(* IEC 61131-3 sources: cc_kush_rewrite/Library, 11 files *)

(* ---- FB_AnalogInput.st ---- *)
FUNCTION_BLOCK FB_AnalogInput
VAR_INPUT
    // Основные входы
    xSimulation     : BOOL;             // Флаг симуляции
    iADC_Code       : INT;              // Код АЦП от модуля аналогового входа
    refEngValue     : REFERENCE TO REAL; // Ссылка на переменную в инженерных единицах
    refSimValue     : REFERENCE TO REAL; // Ссылка на переменную для ручного задания в симуляции

    // Параметры уставок по току (4-20 мА)
    rAlarm_LL       : REAL := 1.1852;      // Аварийно низкий уровень тока (мА)
    rAlarm_L        : REAL := 3.9995;      // Низкий уровень тока (мА)
    rAlarm_H        : REAL := 20.0005;     // Высокий уровень тока (мА)
    rAlarm_HH       : REAL := 22.81;       // Аварийно высокий уровень тока (мА)

    // Параметры АЦП
    iADC_Max        : INT := 32767;     // Максимальный код АЦП
    iADC_Min        : INT := 0;         // Минимальный код АЦП

    // Параметры масштабирования
    rEngValue_Max   : REAL := 100.0;    // Максимальное значение в ед. измерения
    rEngValue_Min   : REAL := 0.0;      // Минимальное значение в ед. измерения

    // Параметры тока
    rCurrent_Max    : REAL := 20.0;     // Максимальный ток (мА)
    rCurrent_Min    : REAL := 4.0;      // Минимальный ток (мА)
END_VAR

VAR_OUTPUT
    // Выходы
    rCurrent_mA     : REAL;             // Ток 4-20 мА

    // Тревоги по току
    xAlarm_LL       : BOOL;             // Аварийно низкий уровень
    xAlarm_L        : BOOL;             // Низкий уровень
    xAlarm_H        : BOOL;             // Высокий уровень
    xAlarm_HH       : BOOL;             // Аварийно высокий уровень
	eAlarmStatus : E_AlarmSetpoints;
END_VAR

VAR
    rScaledValue    : REAL;             // Внутреннее масштабированное значение
    rADC_Range      : REAL;             // Диапазон АЦП
    rEng_Range      : REAL;             // Диапазон инженерных единиц
    rCurrent_Range  : REAL;             // Диапазон тока
    _xSimulation_Prev : BOOL;           // Предыдущее состояние симуляции (для детектирования фронта)
END_VAR

// Расчёт диапазонов
rADC_Range := INT_TO_REAL(iADC_Max - iADC_Min);
rEng_Range := rEngValue_Max - rEngValue_Min;
rCurrent_Range := rCurrent_Max - rCurrent_Min;

// Защита от деления на ноль
IF rADC_Range = 0.0 THEN
    rADC_Range := 1.0;
END_IF

// Масштабирование кода АЦП в ток 4-20 мА
rCurrent_mA := rCurrent_Min +
               (INT_TO_REAL(iADC_Code - iADC_Min) / rADC_Range) * rCurrent_Range;

// Логика симуляции и масштабирования
IF xSimulation THEN
    // Режим симуляции активен

    // При переходе в режим симуляции (rising edge) - инициализировать симуляцию
    IF NOT _xSimulation_Prev AND __ISVALIDREF(refEngValue) AND __ISVALIDREF(refSimValue) THEN
        // Однократно передать текущее значение в переменную симуляции
        refSimValue := refEngValue;
    END_IF

    // В режиме симуляции - использовать значение из переменной симуляции
    IF __ISVALIDREF(refEngValue) AND __ISVALIDREF(refSimValue) THEN
        refEngValue := refSimValue;
    END_IF

ELSE
    // Режим симуляции выключен - работает обычное масштабирование
    IF __ISVALIDREF(refEngValue) THEN
        rScaledValue := rEngValue_Min +
                        ((rCurrent_mA - rCurrent_Min) / rCurrent_Range) * rEng_Range;
        refEngValue := rScaledValue;
    END_IF
END_IF

// Сохранить текущее состояние симуляции для следующего цикла
_xSimulation_Prev := xSimulation;

// Обработка тревог по току
// Аварийно низкий уровень (обрыв линии)
xAlarm_LL := rCurrent_mA < rAlarm_LL;

// Низкий уровень
xAlarm_L := (rCurrent_mA >= rAlarm_LL) AND (rCurrent_mA < rAlarm_L);

// Высокий уровень
xAlarm_H := (rCurrent_mA > rAlarm_H) AND (rCurrent_mA <= rAlarm_HH);

// Аварийно высокий уровень (перегрузка)
xAlarm_HH := rCurrent_mA > rAlarm_HH;

// Обновление общего статуса тревоги (по приоритету)
IF xAlarm_LL THEN
    eAlarmStatus := E_AlarmSetpoints.LL;
ELSIF xAlarm_HH THEN
    eAlarmStatus := E_AlarmSetpoints.HH;
ELSIF xAlarm_L THEN
    eAlarmStatus := E_AlarmSetpoints.L;
ELSIF xAlarm_H THEN
    eAlarmStatus := E_AlarmSetpoints.H;
ELSE
    eAlarmStatus := E_AlarmSetpoints.Normal;
END_IF

END_FUNCTION_BLOCK

(* ---- FB_AnalogOutput.st ---- *)
FUNCTION_BLOCK FB_AnalogOutput
VAR_INPUT
    // Основные входы
    xEnable         : BOOL := TRUE;     // Разрешение работы выхода
    rEngValue       : REAL;             // Значение в инженерных единицах для вывода

    // Параметры масштабирования
    rEngValue_Max   : REAL := 100.0;    // Максимальное значение в ед. измерения
    rEngValue_Min   : REAL := 0.0;      // Минимальное значение в ед. измерения

    // Параметры тока
    rCurrent_Max    : REAL := 20.0;     // Максимальный ток (мА)
    rCurrent_Min    : REAL := 4.0;      // Минимальный ток (мА)

    // Параметры АЦП (DAC)
    iDAC_Max        : INT := 32767;     // Максимальный код АЦП
    iDAC_Min        : INT := 0;         // Минимальный код АЦП

    // Параметры уставок по току (4-20 мА)
    rAlarm_LL       : REAL := 1.1852;      // Аварийно низкий уровень тока (мА)
    rAlarm_L        : REAL := 3.9995;      // Низкий уровень тока (мА)
    rAlarm_H        : REAL := 20.0005;     // Высокий уровень тока (мА)
    rAlarm_HH       : REAL := 22.81;       // Аварийно высокий уровень тока (мА)

    // Опции
    xEnableClamp    : BOOL := TRUE;     // Включить ограничение выхода за пределы диапазона
END_VAR

VAR_OUTPUT
    // Выходы
    rCurrent_mA     : REAL;             // Выходной ток 4-20 мА
    iDAC_Code       : INT;              // Код АЦП для модуля аналогового выхода

    // Тревоги по току
    xAlarm_LL       : BOOL;             // Аварийно низкий уровень
    xAlarm_L        : BOOL;             // Низкий уровень
    xAlarm_H        : BOOL;             // Высокий уровень
    xAlarm_HH       : BOOL;             // Аварийно высокий уровень
    eAlarmStatus    : E_AlarmSetpoints; // Общий статус тревоги

    // Диагностика диапазона
    xOverRange      : BOOL;             // Превышение верхнего предела
    xUnderRange     : BOOL;             // Выход за нижний предел
    xOutOfRange     : BOOL;             // Общий флаг выхода за пределы
END_VAR

VAR
    rEng_Range      : REAL;             // Диапазон инженерных единиц
    rCurrent_Range  : REAL;             // Диапазон тока
    rDAC_Range      : REAL;             // Диапазон АЦП
    rNormalizedValue : REAL;            // Нормализованное значение (0.0 - 1.0)
    rEngValue_Clamped : REAL;           // Ограниченное значение в инженерных единицах
END_VAR

// Расчёт диапазонов
rEng_Range := rEngValue_Max - rEngValue_Min;
rCurrent_Range := rCurrent_Max - rCurrent_Min;
rDAC_Range := INT_TO_REAL(iDAC_Max - iDAC_Min);

// Защита от деления на ноль
IF rEng_Range = 0.0 THEN
    rEng_Range := 1.0;
END_IF

// Проверка выхода за пределы
xUnderRange := rEngValue < rEngValue_Min;
xOverRange := rEngValue > rEngValue_Max;
xOutOfRange := xUnderRange OR xOverRange;

// Ограничение значения (если включено)
IF xEnableClamp THEN
    IF rEngValue < rEngValue_Min THEN
        rEngValue_Clamped := rEngValue_Min;
    ELSIF rEngValue > rEngValue_Max THEN
        rEngValue_Clamped := rEngValue_Max;
    ELSE
        rEngValue_Clamped := rEngValue;
    END_IF
ELSE
    rEngValue_Clamped := rEngValue;
END_IF

// Нормализация значения (0.0 - 1.0)
rNormalizedValue := (rEngValue_Clamped - rEngValue_Min) / rEng_Range;

// Преобразование в ток 4-20 мА
rCurrent_mA := rCurrent_Min + rNormalizedValue * rCurrent_Range;

// Преобразование в код АЦП
IF xEnable THEN
    iDAC_Code := iDAC_Min + REAL_TO_INT(rNormalizedValue * rDAC_Range);
ELSE
    // Если выход отключен - безопасное значение (минимальный ток)
    iDAC_Code := iDAC_Min;
    rCurrent_mA := rCurrent_Min;
END_IF

// Обработка тревог по току
// Аварийно низкий уровень
xAlarm_LL := rCurrent_mA < rAlarm_LL;

// Низкий уровень
xAlarm_L := (rCurrent_mA >= rAlarm_LL) AND (rCurrent_mA < rAlarm_L);

// Высокий уровень
xAlarm_H := (rCurrent_mA > rAlarm_H) AND (rCurrent_mA <= rAlarm_HH);

// Аварийно высокий уровень
xAlarm_HH := rCurrent_mA > rAlarm_HH;

// Обновление общего статуса тревоги (по приоритету)
IF xAlarm_LL THEN
    eAlarmStatus := E_AlarmSetpoints.LL;
ELSIF xAlarm_HH THEN
    eAlarmStatus := E_AlarmSetpoints.HH;
ELSIF xAlarm_L THEN
    eAlarmStatus := E_AlarmSetpoints.L;
ELSIF xAlarm_H THEN
    eAlarmStatus := E_AlarmSetpoints.H;
ELSE
    eAlarmStatus := E_AlarmSetpoints.Normal;
END_IF

END_FUNCTION_BLOCK

(* ---- FB_FrequencyControl.st ---- *)
FUNCTION_BLOCK FB_FrequencyControl
VAR_INPUT
    irMaxFrequency : REAL := 100.0;             // Максимальная частота
    irStep : REAL := 1.0;                       // Шаг изменения частоты по умолчанию
    rTargetFrequency : REAL := 0.0;             // Целевая частота (уставка)
    xPulse : BOOL;                              // Импульсный сигнал для вычисления
    xConditionToProceed : BOOL := TRUE;         // Условия для продолжения вычисления
    xReset : BOOL;                              // Сброс частоты в ноль
    xHold : BOOL;                               // Удержание текущей частоты
END_VAR
VAR_OUTPUT
    qrCurrentFrequency : REAL;                  // Текущая выходная частота
    qrTargetFrequency : REAL;                   // Целевая частота
    qxTargetReached : BOOL;                     // Флаг достижения целевой частоты
END_VAR
VAR
    _rSetFrequency : REAL;                      // Целевая частота (уставка) внутренняя
    _rCurrentFrequency : REAL;                  // Текущая частота (внутренняя)
    _xInitialized : BOOL := FALSE;              // Флаг инициализации
END_VAR

// Инициализация при первом вызове
IF NOT _xInitialized THEN
    _rCurrentFrequency := 0.0;
    _rSetFrequency := 0.0;
    _xInitialized := TRUE;
END_IF

// Сброс частоты
IF xReset THEN
    _rCurrentFrequency := 0.0;
    _rSetFrequency := 0.0;
    qrCurrentFrequency := 0.0;
    qrTargetFrequency := 0.0;
    qxTargetReached := TRUE;
    RETURN;
END_IF

// Удержание текущей частоты
IF xHold THEN
    _rSetFrequency := _rCurrentFrequency;
    qxTargetReached := TRUE;
END_IF

// Обновление целевой частоты
_rSetFrequency := rTargetFrequency;

// Ограничение целевой частоты
IF _rSetFrequency > irMaxFrequency THEN
    _rSetFrequency := irMaxFrequency;
ELSIF _rSetFrequency < 0.0 THEN
    _rSetFrequency := 0.0;
END_IF

// Обработка изменения частоты
IF xPulse AND xConditionToProceed THEN
    // Плавное изменение частоты к уставке
    IF _rCurrentFrequency < _rSetFrequency - irStep THEN
        // Увеличиваем частоту
        _rCurrentFrequency := _rCurrentFrequency + irStep;
        qxTargetReached := FALSE;
    ELSIF _rCurrentFrequency > _rSetFrequency + irStep THEN
        // Уменьшаем частоту
        _rCurrentFrequency := _rCurrentFrequency - irStep;
        qxTargetReached := FALSE;
    ELSE
        // Достигли целевой частоты
        _rCurrentFrequency := _rSetFrequency;
        qxTargetReached := TRUE;
    END_IF
ELSE
    // Проверяем, достигнута ли целевая частота
    IF ABS(_rCurrentFrequency - _rSetFrequency) < 0.01 THEN
        qxTargetReached := TRUE;
    ELSE
        qxTargetReached := FALSE;
    END_IF
END_IF

// Обновляем выходные значения
qrCurrentFrequency := _rCurrentFrequency;
qrTargetFrequency := _rSetFrequency;

END_FUNCTION_BLOCK

(* ---- FB_NumericChangeDetector.st ---- *)
FUNCTION_BLOCK FB_NumericChangeDetector
VAR_INPUT
    irValue : REAL;                             // Входное числовое значение для мониторинга
    xReset : BOOL;                              // Сброс детектора изменений
END_VAR
VAR_OUTPUT
    qxChangeDetected : BOOL;                    // Импульс при обнаружении изменения значения
    qrCurrentValue : REAL;                      // Текущее отслеживаемое значение
    qrPreviousValue : REAL;                     // Предыдущее значение
    qrValueDifference : REAL;                   // Разность между текущим и предыдущим значением
    qxValueIncreased : BOOL;                    // Флаг увеличения значения
    qxValueDecreased : BOOL;                    // Флаг уменьшения значения
END_VAR
VAR
    _rPreviousValue : REAL := 0.0;              // Предыдущее значение для сравнения
    _xFirstCycle : BOOL := TRUE;                // Флаг первого цикла выполнения
    _rt_Change : R_TRIG;                        // Триггер для генерации импульса
    _xValueChanged : BOOL := FALSE;             // Внутренний флаг изменения
END_VAR

// Сброс детектора
IF xReset THEN
    _rPreviousValue := irValue;
    _xFirstCycle := TRUE;
    _xValueChanged := FALSE;
    _rt_Change(CLK := FALSE);
    qxChangeDetected := FALSE;
    qrValueDifference := 0.0;
    qxValueIncreased := FALSE;
    qxValueDecreased := FALSE;
    RETURN;
END_IF

// Пропускаем первый цикл для корректной инициализации
IF _xFirstCycle THEN
    _rPreviousValue := irValue;
    _xFirstCycle := FALSE;
    _xValueChanged := FALSE;
ELSE
    // Проверяем изменение значения
    IF _rPreviousValue <> irValue THEN
        _xValueChanged := TRUE;
    ELSE
        _xValueChanged := FALSE;
    END_IF
END_IF

// Генерируем импульс при изменении через R_TRIG
_rt_Change(CLK := _xValueChanged);
qxChangeDetected := _rt_Change.Q;

// Вычисляем разность
qrValueDifference := irValue - _rPreviousValue;

// Определяем направление изменения
qxValueIncreased := _xValueChanged AND (irValue > _rPreviousValue);
qxValueDecreased := _xValueChanged AND (irValue < _rPreviousValue);

// Обновляем предыдущее значение после всех вычислений
IF _xValueChanged THEN
    _rPreviousValue := irValue;
END_IF

// Обновляем выходы
qrCurrentValue := irValue;
qrPreviousValue := _rPreviousValue;

END_FUNCTION_BLOCK

(* ---- FB_PreStartAlarm.st ---- *)
FUNCTION_BLOCK FB_PreStartAlarm
VAR_INPUT
    ixStart : BOOL;                    // Сигнал на запуск
    ixStop : BOOL;                     // Сигнал на стоп (Reset)
    itFirstSignal : TIME;              // Уставка первого сигнала
    itPauseAfterFirst : TIME;          // Уставка паузы после первого сигнала
    itSecondSignal : TIME;             // Уставка второго сигнала
    itPauseAfterSecond : TIME;         // Уставка паузы после второго сигнала
END_VAR

VAR_OUTPUT
    qxAlarmPower : BOOL;               // Питание звуковой сигнализации
    qxActive : BOOL;                   // Активная работа ФБ
    qxComplete : BOOL;                 // Импульс о завершении работы
    qnSecondsRemaining : INT;          // Количество секунд до завершения
    qwSecondsRemaining : WORD;		    // Количество секунд до завершения (тип WORD)
END_VAR

VAR
    _eState : (
        IDLE := 0,              // Ожидание запуска
        FIRST_SIGNAL := 1,      // Первый звуковой сигнал
        PAUSE_AFTER_FIRST := 2, // Пауза после первого сигнала
        SECOND_SIGNAL := 3,     // Второй звуковой сигнал
        PAUSE_AFTER_SECOND := 4,// Пауза после второго сигнала
        COMPLETE := 5           // Завершение
    ) := IDLE;                         // Состояние автомата
    _tonTimer : TON;                   // Универсальный таймер для всех этапов
    _xCompleteInternal : BOOL;         // Внутренний сигнал завершения
    _rtrigComplete : R_TRIG;           // Детектор переднего фронта для импульса завершения
END_VAR

qwSecondsRemaining := TO_WORD(qnSecondsRemaining);

// Обработка сигнала СТОП (сброс)
IF ixStop THEN
    _eState := IDLE;
    qxActive := FALSE;
    qxAlarmPower := FALSE;
    _tonTimer(IN := FALSE);
    _xCompleteInternal := FALSE;
    qxComplete := FALSE;
    qnSecondsRemaining := 0;
    RETURN;
END_IF

// Автомат состояний
CASE _eState OF

    IDLE: // Ожидание запуска
        qxActive := FALSE;
        qxAlarmPower := FALSE;
        _xCompleteInternal := FALSE;
        _tonTimer(IN := FALSE);
        qnSecondsRemaining := 0;

        IF ixStart THEN
			qxActive := TRUE;
            _eState := FIRST_SIGNAL;
        END_IF

    FIRST_SIGNAL: // Первый сигнал
        qxAlarmPower := TRUE;
        _tonTimer(IN := TRUE, PT := itFirstSignal);

        // Расчет оставшегося времени в секундах
        qnSecondsRemaining := DINT_TO_INT(
            (TIME_TO_DINT(itFirstSignal - _tonTimer.ET) +
             TIME_TO_DINT(itPauseAfterFirst) +
             TIME_TO_DINT(itSecondSignal) +
             TIME_TO_DINT(itPauseAfterSecond)) / 1000
        );

        IF _tonTimer.Q THEN
            _tonTimer(IN := FALSE);
            _eState := PAUSE_AFTER_FIRST;
        END_IF

    PAUSE_AFTER_FIRST: // Пауза после первого сигнала
        qxAlarmPower := FALSE;
        _tonTimer(IN := TRUE, PT := itPauseAfterFirst);

        // Расчет оставшегося времени в секундах
        qnSecondsRemaining := DINT_TO_INT(
            (TIME_TO_DINT(itPauseAfterFirst - _tonTimer.ET) +
             TIME_TO_DINT(itSecondSignal) +
             TIME_TO_DINT(itPauseAfterSecond)) / 1000
        );

        IF _tonTimer.Q THEN
            _tonTimer(IN := FALSE);
            _eState := SECOND_SIGNAL;
        END_IF

    SECOND_SIGNAL: // Второй сигнал
        qxAlarmPower := TRUE;
        _tonTimer(IN := TRUE, PT := itSecondSignal);

        // Расчет оставшегося времени в секундах
        qnSecondsRemaining := DINT_TO_INT(
            (TIME_TO_DINT(itSecondSignal - _tonTimer.ET) +
             TIME_TO_DINT(itPauseAfterSecond)) / 1000
        );

        IF _tonTimer.Q THEN
            _tonTimer(IN := FALSE);
            _eState := PAUSE_AFTER_SECOND;
        END_IF

    PAUSE_AFTER_SECOND: // Пауза после второго сигнала
        qxAlarmPower := FALSE;
        _tonTimer(IN := TRUE, PT := itPauseAfterSecond);

        // Расчет оставшегося времени в секундах
        qnSecondsRemaining := DINT_TO_INT(
            TIME_TO_DINT(itPauseAfterSecond - _tonTimer.ET) / 1000
        );

        IF _tonTimer.Q THEN
            _tonTimer(IN := FALSE);
            _eState := COMPLETE;
        END_IF

    COMPLETE: // Завершение
        qxAlarmPower := FALSE;
        qxActive := FALSE;
        _xCompleteInternal := TRUE;
        qnSecondsRemaining := 0;
        _eState := IDLE;  // Вернуться в начальное состояние
END_CASE

// Генерация импульса завершения через R_TRIG
_rtrigComplete(CLK := _xCompleteInternal);
qxComplete := _rtrigComplete.Q;

END_FUNCTION_BLOCK

(* ---- FB_ProportionPID.st ---- *)
FUNCTION_BLOCK FB_ProportionPID

// ============================================================================
// ВХОДНЫЕ ПЕРЕМЕННЫЕ
// ============================================================================
VAR_INPUT
    // ------------------------------------------------------------------------
    // Команды управления
    // ------------------------------------------------------------------------
    xEnable                 : BOOL;         // Разрешение работы блока
    xReset                  : BOOL;         // Сброс интегральной составляющей ПИД

    // ------------------------------------------------------------------------
    // Целевые пропорции (уставки оператора)
    // ------------------------------------------------------------------------
    rProportionTarget_1     : REAL;         // Целевая пропорция бункера 1 [0..1]
    rProportionTarget_2     : REAL;         // Целевая пропорция бункера 2 [0..1]
    rProportionTarget_3     : REAL;         // Целевая пропорция бункера 3 [0..1]
                                            // Сумма должна = 1.0 (100%)
                                            // Значение 0.0 = бункер неактивен

    // ------------------------------------------------------------------------
    // Фактические пропорции (с конвейерных весов)
    // ------------------------------------------------------------------------
    rProportionActual_1     : REAL;         // Фактическая пропорция бункера 1 [0..1]
    rProportionActual_2     : REAL;         // Фактическая пропорция бункера 2 [0..1]
    rProportionActual_3     : REAL;         // Фактическая пропорция бункера 3 [0..1]

    // ------------------------------------------------------------------------
    // Параметры ПИД-регулятора
    // ------------------------------------------------------------------------
    rPID_Kp                 : REAL := 1.0;  // Пропорциональный коэффициент
    rPID_Ki                 : REAL := 0.2;  // Интегральный коэффициент
    rPID_Kd                 : REAL := 0.05; // Дифференциальный коэффициент
    rPID_IntegralLimit      : REAL := 10.0; // Ограничение интеграла (anti-windup)
    rPID_DerivativeFilter   : REAL := 0.1;  // Коэффициент фильтрации D-составляющей [0..1]
                                            // 0 = нет фильтрации, 1 = максимум фильтра

    // ------------------------------------------------------------------------
    // Базовые частоты (рассчитываются заранее в INIT)
    // ------------------------------------------------------------------------
    rFrequencyBase_1        : REAL;         // Базовая частота бункера 1, Гц
    rFrequencyBase_2        : REAL;         // Базовая частота бункера 2, Гц
    rFrequencyBase_3        : REAL;         // Базовая частота бункера 3, Гц

    // ------------------------------------------------------------------------
    // Параметры оборудования
    // ------------------------------------------------------------------------
    rFrequency_Min          : REAL := 1.0;  // Минимальная частота ЧРП, Гц
    rFrequency_Max          : REAL := 35.0; // Максимальная частота ЧРП, Гц
    rFrequency_TargetSum    : REAL := 90.0; // Целевая суммарная частота для нормализации, Гц

    // ------------------------------------------------------------------------
    // Параметры расчета
    // ------------------------------------------------------------------------
    rDeltaTime              : REAL := 2;  // Период вызова блока, сек

    // ------------------------------------------------------------------------
    // Параметры алгоритма
    // ------------------------------------------------------------------------
    rScaleLimit_Min         : REAL := 0.1;  // Минимальный коэффициент масштабирования
    rScaleLimit_Max         : REAL := 3.0;  // Максимальный коэффициент масштабирования
    rProportionThreshold    : REAL := 0.001; // Порог для определения неактивного бункера
END_VAR

// ============================================================================
// ВЫХОДНЫЕ ПЕРЕМЕННЫЕ
// ============================================================================
VAR_OUTPUT
    // ------------------------------------------------------------------------
    // Управляющие воздействия (частоты ЧРП)
    // ------------------------------------------------------------------------
    qrFrequency_1           : REAL;         // Уставка частоты ЧРП бункера 1, Гц
    qrFrequency_2           : REAL;         // Уставка частоты ЧРП бункера 2, Гц
    qrFrequency_3           : REAL;         // Уставка частоты ЧРП бункера 3, Гц

    // ------------------------------------------------------------------------
    // Состояние работы
    // ------------------------------------------------------------------------
    qxActive                : BOOL;         // Блок активен и регулирует частоты
    qxError                 : BOOL;         // Ошибка работы блока
    quErrorCode             : UINT;         // Код ошибки:
                                            // 0 = нет ошибок
                                            // 1 = сумма пропорций = 0
                                            // 2 = неверный DeltaTime
                                            // 3 = неверные пределы частот
                                            // 4 = неверная целевая сумма частот

    // ------------------------------------------------------------------------
    // Диагностическая информация
    // ------------------------------------------------------------------------
    qrFrequency_Sum         : REAL;         // Фактическая суммарная частота, Гц
    qrProportionSum         : REAL;         // Сумма целевых пропорций
    qxProportionNormalized  : BOOL;         // TRUE = пропорции автоматически нормализованы

    // ------------------------------------------------------------------------
    // Выходы ПИД-регуляторов (для диагностики)
    // ------------------------------------------------------------------------
    qrPID_Output_1          : REAL;         // Выход ПИД регулятора 1 [0..1]
    qrPID_Output_2          : REAL;         // Выход ПИД регулятора 2 [0..1]
    qrPID_Output_3          : REAL;         // Выход ПИД регулятора 3 [0..1]

    qrPID_Error_1           : REAL;         // Текущая ошибка ПИД 1
    qrPID_Error_2           : REAL;         // Текущая ошибка ПИД 2
    qrPID_Error_3           : REAL;         // Текущая ошибка ПИД 3

    qrPID_Integral_1        : REAL;         // Интегральная составляющая ПИД 1
    qrPID_Integral_2        : REAL;         // Интегральная составляющая ПИД 2
    qrPID_Integral_3        : REAL;         // Интегральная составляющая ПИД 3
END_VAR

// ============================================================================
// ВНУТРЕННИЕ ПЕРЕМЕННЫЕ
// ============================================================================
VAR
    // ------------------------------------------------------------------------
    // Состояние ПИД-регуляторов
    // ------------------------------------------------------------------------
    _rPrevError_1           : REAL := 0.0;  // Предыдущая ошибка ПИД 1
    _rPrevError_2           : REAL := 0.0;  // Предыдущая ошибка ПИД 2
    _rPrevError_3           : REAL := 0.0;  // Предыдущая ошибка ПИД 3

    _rIntegral_1            : REAL := 0.0;  // Интегральная составляющая ПИД 1
    _rIntegral_2            : REAL := 0.0;  // Интегральная составляющая ПИД 2
    _rIntegral_3            : REAL := 0.0;  // Интегральная составляющая ПИД 3

    _rDerivativeFiltered_1  : REAL := 0.0;  // Фильтрованная производная ПИД 1
    _rDerivativeFiltered_2  : REAL := 0.0;  // Фильтрованная производная ПИД 2
    _rDerivativeFiltered_3  : REAL := 0.0;  // Фильтрованная производная ПИД 3

    // ------------------------------------------------------------------------
    // Флаги активности бункеров
    // ------------------------------------------------------------------------
    _xBunker1_Active        : BOOL := FALSE; // Бункер 1 активен
    _xBunker2_Active        : BOOL := FALSE; // Бункер 2 активен
    _xBunker3_Active        : BOOL := FALSE; // Бункер 3 активен

    // ------------------------------------------------------------------------
    // Нормализованные пропорции
    // ------------------------------------------------------------------------
    _rProportionNorm_1      : REAL := 0.0;  // Нормализованная пропорция 1
    _rProportionNorm_2      : REAL := 0.0;  // Нормализованная пропорция 2
    _rProportionNorm_3      : REAL := 0.0;  // Нормализованная пропорция 3

    // ------------------------------------------------------------------------
    // Промежуточные расчеты частот
    // ------------------------------------------------------------------------
    _rFreqScaled_1          : REAL := 0.0;  // Масштабированная частота 1
    _rFreqScaled_2          : REAL := 0.0;  // Масштабированная частота 2
    _rFreqScaled_3          : REAL := 0.0;  // Масштабированная частота 3

    _rScale_1               : REAL := 1.0;  // Коэффициент масштабирования 1
    _rScale_2               : REAL := 1.0;  // Коэффициент масштабирования 2
    _rScale_3               : REAL := 1.0;  // Коэффициент масштабирования 3

    // ------------------------------------------------------------------------
    // Вспомогательные переменные
    // ------------------------------------------------------------------------
    _rError                 : REAL;         // Текущая ошибка (временная)
    _rDerivative            : REAL;         // Дифференциальная составляющая (временная)
    _rOutput                : REAL;         // Выход ПИД (временная)
    _rSumScaled             : REAL;         // Сумма масштабированных частот
    _rProportionSumInput    : REAL;         // Сумма входных пропорций
END_VAR

// ============================================================================
// ОСНОВНОЙ КОД ФУНКЦИОНАЛЬНОГО БЛОКА
// ============================================================================

// ============================================================================
// ПРОВЕРКА КОМАНДЫ ENABLE
// ============================================================================
IF NOT xEnable THEN
    // Блок выключен - сброс всех выходов
    qxActive := FALSE;
    qrFrequency_1 := 0.0;
    qrFrequency_2 := 0.0;
    qrFrequency_3 := 0.0;
    qrFrequency_Sum := 0.0;

    // Сброс диагностических выходов
    qrPID_Output_1 := 0.0;
    qrPID_Output_2 := 0.0;
    qrPID_Output_3 := 0.0;
    qrPID_Error_1 := 0.0;
    qrPID_Error_2 := 0.0;
    qrPID_Error_3 := 0.0;
    qrPID_Integral_1 := 0.0;
    qrPID_Integral_2 := 0.0;
    qrPID_Integral_3 := 0.0;

    // Сброс внутренних переменных ПИД
    _rIntegral_1 := 0.0;
    _rIntegral_2 := 0.0;
    _rIntegral_3 := 0.0;
    _rPrevError_1 := 0.0;
    _rPrevError_2 := 0.0;
    _rPrevError_3 := 0.0;
    _rDerivativeFiltered_1 := 0.0;
    _rDerivativeFiltered_2 := 0.0;
    _rDerivativeFiltered_3 := 0.0;

    RETURN; // Выход из блока
END_IF

// ============================================================================
// ВАЛИДАЦИЯ ПАРАМЕТРОВ И ДИАГНОСТИКА ОШИБОК
// ============================================================================
qxError := FALSE;
quErrorCode := 0;

// Проверка периода вызова
IF rDeltaTime <= 0.0 OR rDeltaTime > 1.0 THEN
    qxError := TRUE;
    quErrorCode := 2;
    RETURN;
END_IF

// Проверка пределов частот
IF rFrequency_Min >= rFrequency_Max THEN
    qxError := TRUE;
    quErrorCode := 3;
    RETURN;
END_IF

// Проверка целевой суммы частот
IF rFrequency_TargetSum <= 0.0 THEN
    qxError := TRUE;
    quErrorCode := 4;
    RETURN;
END_IF

// ============================================================================
// ВАЛИДАЦИЯ И НОРМАЛИЗАЦИЯ ЦЕЛЕВЫХ ПРОПОРЦИЙ
// ============================================================================
_rProportionSumInput := rProportionTarget_1 + rProportionTarget_2 + rProportionTarget_3;

// Проверка: сумма пропорций должна быть > 0
IF _rProportionSumInput < 0.0001 THEN
    // Все бункеры неактивны
    qxError := TRUE;
    quErrorCode := 1;
    qrFrequency_1 := 0.0;
    qrFrequency_2 := 0.0;
    qrFrequency_3 := 0.0;
    qrFrequency_Sum := 0.0;
    RETURN;
END_IF

// Нормализация пропорций, если сумма != 1.0
IF ABS(_rProportionSumInput - 1.0) > 0.001 THEN
    _rProportionNorm_1 := rProportionTarget_1 / _rProportionSumInput;
    _rProportionNorm_2 := rProportionTarget_2 / _rProportionSumInput;
    _rProportionNorm_3 := rProportionTarget_3 / _rProportionSumInput;
    qxProportionNormalized := TRUE;
ELSE
    _rProportionNorm_1 := rProportionTarget_1;
    _rProportionNorm_2 := rProportionTarget_2;
    _rProportionNorm_3 := rProportionTarget_3;
    qxProportionNormalized := FALSE;
END_IF

qrProportionSum := _rProportionNorm_1 + _rProportionNorm_2 + _rProportionNorm_3;

// ============================================================================
// ОПРЕДЕЛЕНИЕ АКТИВНОСТИ БУНКЕРОВ
// ============================================================================
_xBunker1_Active := (_rProportionNorm_1 > rProportionThreshold);
_xBunker2_Active := (_rProportionNorm_2 > rProportionThreshold);
_xBunker3_Active := (_rProportionNorm_3 > rProportionThreshold);

// ============================================================================
// ОБРАБОТКА КОМАНДЫ RESET (сброс интегралов)
// ============================================================================
IF xReset THEN
    _rIntegral_1 := 0.0;
    _rIntegral_2 := 0.0;
    _rIntegral_3 := 0.0;
    _rPrevError_1 := 0.0;
    _rPrevError_2 := 0.0;
    _rPrevError_3 := 0.0;
END_IF

// ============================================================================
// ОБНОВЛЕНИЕ ПИД-РЕГУЛЯТОРОВ
// ============================================================================

// ----------------------------------------------------------------------------
// ПИД-регулятор бункера 1
// ----------------------------------------------------------------------------
IF _xBunker1_Active THEN
    // Расчет ошибки регулирования
    _rError := _rProportionNorm_1 - rProportionActual_1;
    qrPID_Error_1 := _rError;

    // Расчет дифференциальной составляющей (сырая производная)
    _rDerivative := (_rError - _rPrevError_1) / rDeltaTime;

    // Низкочастотный фильтр первого порядка для D-составляющей
    // D_filtered(n) = alpha * D_raw + (1-alpha) * D_filtered(n-1)
    // alpha = 1 - rPID_DerivativeFilter (меньше alpha = больше фильтрации)
    _rDerivativeFiltered_1 := (1.0 - rPID_DerivativeFilter) * _rDerivative
                            + rPID_DerivativeFilter * _rDerivativeFiltered_1;

    // ПИД формула: u(t) = Kp*e(t) + Ki*∫e(t)dt + Kd*de(t)/dt
    _rOutput := rPID_Kp * _rError + rPID_Ki * _rIntegral_1 + rPID_Kd * _rDerivativeFiltered_1;

    // Условная интеграция (conditional integration anti-windup):
    // Накапливаем интеграл ТОЛЬКО если выход не насыщен
    // или если ошибка уменьшает насыщение
    IF (_rOutput >= 0.0 AND _rOutput <= 1.0) OR
       (_rOutput < 0.0 AND _rError > 0.0) OR
       (_rOutput > 1.0 AND _rError < 0.0) THEN
        _rIntegral_1 := _rIntegral_1 + _rError * rDeltaTime;

        // Ограничение интеграла (дополнительная защита)
        IF _rIntegral_1 > rPID_IntegralLimit THEN
            _rIntegral_1 := rPID_IntegralLimit;
        ELSIF _rIntegral_1 < -rPID_IntegralLimit THEN
            _rIntegral_1 := -rPID_IntegralLimit;
        END_IF
    END_IF

    qrPID_Integral_1 := _rIntegral_1;

    // Ограничение выхода в диапазоне [0..1]
    IF _rOutput < 0.0 THEN
        _rOutput := 0.0;
    ELSIF _rOutput > 1.0 THEN
        _rOutput := 1.0;
    END_IF

    qrPID_Output_1 := _rOutput;

    // Сохранение ошибки для следующей итерации
    _rPrevError_1 := _rError;
ELSE
    // Бункер неактивен - сброс ПИД
    qrPID_Output_1 := 0.0;
    qrPID_Error_1 := 0.0;
    qrPID_Integral_1 := 0.0;
    _rIntegral_1 := 0.0;              // КРИТИЧНО: сброс внутреннего интеграла
    _rPrevError_1 := 0.0;
    _rDerivativeFiltered_1 := 0.0;    // Сброс фильтра производной
END_IF

// ----------------------------------------------------------------------------
// ПИД-регулятор бункера 2
// ----------------------------------------------------------------------------
IF _xBunker2_Active THEN
    _rError := _rProportionNorm_2 - rProportionActual_2;
    qrPID_Error_2 := _rError;

    _rDerivative := (_rError - _rPrevError_2) / rDeltaTime;
    _rDerivativeFiltered_2 := (1.0 - rPID_DerivativeFilter) * _rDerivative
                            + rPID_DerivativeFilter * _rDerivativeFiltered_2;

    _rOutput := rPID_Kp * _rError + rPID_Ki * _rIntegral_2 + rPID_Kd * _rDerivativeFiltered_2;

    // Условная интеграция (anti-windup)
    IF (_rOutput >= 0.0 AND _rOutput <= 1.0) OR
       (_rOutput < 0.0 AND _rError > 0.0) OR
       (_rOutput > 1.0 AND _rError < 0.0) THEN
        _rIntegral_2 := _rIntegral_2 + _rError * rDeltaTime;

        IF _rIntegral_2 > rPID_IntegralLimit THEN
            _rIntegral_2 := rPID_IntegralLimit;
        ELSIF _rIntegral_2 < -rPID_IntegralLimit THEN
            _rIntegral_2 := -rPID_IntegralLimit;
        END_IF
    END_IF

    qrPID_Integral_2 := _rIntegral_2;

    IF _rOutput < 0.0 THEN
        _rOutput := 0.0;
    ELSIF _rOutput > 1.0 THEN
        _rOutput := 1.0;
    END_IF

    qrPID_Output_2 := _rOutput;
    _rPrevError_2 := _rError;
ELSE
    qrPID_Output_2 := 0.0;
    qrPID_Error_2 := 0.0;
    qrPID_Integral_2 := 0.0;
    _rIntegral_2 := 0.0;              // КРИТИЧНО: сброс внутреннего интеграла
    _rPrevError_2 := 0.0;
    _rDerivativeFiltered_2 := 0.0;    // Сброс фильтра производной
END_IF

// ----------------------------------------------------------------------------
// ПИД-регулятор бункера 3
// ----------------------------------------------------------------------------
IF _xBunker3_Active THEN
    _rError := _rProportionNorm_3 - rProportionActual_3;
    qrPID_Error_3 := _rError;

    _rDerivative := (_rError - _rPrevError_3) / rDeltaTime;
    _rDerivativeFiltered_3 := (1.0 - rPID_DerivativeFilter) * _rDerivative
                            + rPID_DerivativeFilter * _rDerivativeFiltered_3;

    _rOutput := rPID_Kp * _rError + rPID_Ki * _rIntegral_3 + rPID_Kd * _rDerivativeFiltered_3;

    // Условная интеграция (anti-windup)
    IF (_rOutput >= 0.0 AND _rOutput <= 1.0) OR
       (_rOutput < 0.0 AND _rError > 0.0) OR
       (_rOutput > 1.0 AND _rError < 0.0) THEN
        _rIntegral_3 := _rIntegral_3 + _rError * rDeltaTime;

        IF _rIntegral_3 > rPID_IntegralLimit THEN
            _rIntegral_3 := rPID_IntegralLimit;
        ELSIF _rIntegral_3 < -rPID_IntegralLimit THEN
            _rIntegral_3 := -rPID_IntegralLimit;
        END_IF
    END_IF

    qrPID_Integral_3 := _rIntegral_3;

    IF _rOutput < 0.0 THEN
        _rOutput := 0.0;
    ELSIF _rOutput > 1.0 THEN
        _rOutput := 1.0;
    END_IF

    qrPID_Output_3 := _rOutput;
    _rPrevError_3 := _rError;
ELSE
    qrPID_Output_3 := 0.0;
    qrPID_Error_3 := 0.0;
    qrPID_Integral_3 := 0.0;
    _rIntegral_3 := 0.0;              // КРИТИЧНО: сброс внутреннего интеграла
    _rPrevError_3 := 0.0;
    _rDerivativeFiltered_3 := 0.0;    // Сброс фильтра производной
END_IF

// ============================================================================
// РАСЧЕТ ЧАСТОТ ЧРП (АДАПТИВНЫЙ АЛГОРИТМ)
// ============================================================================
// Базовые частоты (rFrequencyBase_1/2/3) рассчитываются заранее в INIT
// на основе пропорций и целевой суммарной частоты

// ----------------------------------------------------------------------------
// ШАГ 1: Применение ПИД-коррекции к базовым частотам
// ----------------------------------------------------------------------------
// Новый алгоритм: ПИД-выход напрямую добавляется к базовой частоте
// Формула: Freq = FreqBase + PID_Output * CorrectioRange
// где CorrectionRange = диапазон коррекции вокруг базовой частоты

// Бункер 1
IF _xBunker1_Active THEN
    // Диапазон коррекции = базовая частота (можно изменить на другой коэффициент)
    _rScale_1 := rFrequencyBase_1;

    // ПИД-выход [0..1] преобразуется в коррекцию [-FreqBase..+FreqBase]
    // qrPID_Output_1 = 0.5 → нет коррекции
    // qrPID_Output_1 > 0.5 → увеличение частоты
    // qrPID_Output_1 < 0.5 → уменьшение частоты
    _rFreqScaled_1 := rFrequencyBase_1 + (qrPID_Output_1 - 0.5) * 2.0 * _rScale_1;

    // Ограничение коэффициента масштабирования (для диагностики)
    _rScale_1 := _rFreqScaled_1 / rFrequencyBase_1;
    IF _rScale_1 < rScaleLimit_Min THEN
        _rScale_1 := rScaleLimit_Min;
        _rFreqScaled_1 := rFrequencyBase_1 * _rScale_1;
    ELSIF _rScale_1 > rScaleLimit_Max THEN
        _rScale_1 := rScaleLimit_Max;
        _rFreqScaled_1 := rFrequencyBase_1 * _rScale_1;
    END_IF
ELSE
    _rFreqScaled_1 := 0.0;
    _rScale_1 := 0.0;
END_IF

// Бункер 2
IF _xBunker2_Active THEN
    _rScale_2 := rFrequencyBase_2;
    _rFreqScaled_2 := rFrequencyBase_2 + (qrPID_Output_2 - 0.5) * 2.0 * _rScale_2;

    _rScale_2 := _rFreqScaled_2 / rFrequencyBase_2;
    IF _rScale_2 < rScaleLimit_Min THEN
        _rScale_2 := rScaleLimit_Min;
        _rFreqScaled_2 := rFrequencyBase_2 * _rScale_2;
    ELSIF _rScale_2 > rScaleLimit_Max THEN
        _rScale_2 := rScaleLimit_Max;
        _rFreqScaled_2 := rFrequencyBase_2 * _rScale_2;
    END_IF
ELSE
    _rFreqScaled_2 := 0.0;
    _rScale_2 := 0.0;
END_IF

// Бункер 3
IF _xBunker3_Active THEN
    _rScale_3 := rFrequencyBase_3;
    _rFreqScaled_3 := rFrequencyBase_3 + (qrPID_Output_3 - 0.5) * 2.0 * _rScale_3;

    _rScale_3 := _rFreqScaled_3 / rFrequencyBase_3;
    IF _rScale_3 < rScaleLimit_Min THEN
        _rScale_3 := rScaleLimit_Min;
        _rFreqScaled_3 := rFrequencyBase_3 * _rScale_3;
    ELSIF _rScale_3 > rScaleLimit_Max THEN
        _rScale_3 := rScaleLimit_Max;
        _rFreqScaled_3 := rFrequencyBase_3 * _rScale_3;
    END_IF
ELSE
    _rFreqScaled_3 := 0.0;
    _rScale_3 := 0.0;
END_IF

// ----------------------------------------------------------------------------
// ШАГ 2: Применение ограничений оборудования (до нормализации!)
// ----------------------------------------------------------------------------

// Бункер 1
IF _xBunker1_Active THEN
    IF _rFreqScaled_1 > rFrequency_Max THEN
        _rFreqScaled_1 := rFrequency_Max;
    ELSIF _rFreqScaled_1 < rFrequency_Min THEN
        _rFreqScaled_1 := rFrequency_Min;
    END_IF
ELSE
    _rFreqScaled_1 := 0.0;
END_IF

// Бункер 2
IF _xBunker2_Active THEN
    IF _rFreqScaled_2 > rFrequency_Max THEN
        _rFreqScaled_2 := rFrequency_Max;
    ELSIF _rFreqScaled_2 < rFrequency_Min THEN
        _rFreqScaled_2 := rFrequency_Min;
    END_IF
ELSE
    _rFreqScaled_2 := 0.0;
END_IF

// Бункер 3
IF _xBunker3_Active THEN
    IF _rFreqScaled_3 > rFrequency_Max THEN
        _rFreqScaled_3 := rFrequency_Max;
    ELSIF _rFreqScaled_3 < rFrequency_Min THEN
        _rFreqScaled_3 := rFrequency_Min;
    END_IF
ELSE
    _rFreqScaled_3 := 0.0;
END_IF

// ----------------------------------------------------------------------------
// ШАГ 3: Нормализация для поддержания целевой суммарной частоты
// ----------------------------------------------------------------------------
// КРИТИЧНО: нормализация ПОСЛЕ ограничений, чтобы сумма всегда = TargetSum
_rSumScaled := _rFreqScaled_1 + _rFreqScaled_2 + _rFreqScaled_3;

// Защита от деления на ноль
IF _rSumScaled < 0.01 THEN
    _rSumScaled := 0.01;
END_IF

qrFrequency_1 := _rFreqScaled_1 * (rFrequency_TargetSum / _rSumScaled);
qrFrequency_2 := _rFreqScaled_2 * (rFrequency_TargetSum / _rSumScaled);
qrFrequency_3 := _rFreqScaled_3 * (rFrequency_TargetSum / _rSumScaled);

// ============================================================================
// ОБНОВЛЕНИЕ ДИАГНОСТИЧЕСКИХ ВЫХОДОВ
// ============================================================================
qrFrequency_Sum := qrFrequency_1 + qrFrequency_2 + qrFrequency_3;
qxActive := TRUE;

END_FUNCTION_BLOCK

(* ---- FB_RangeDiagnostic.st ---- *)
FUNCTION_BLOCK FB_RangeDiagnostic
VAR_INPUT
    irValue : REAL;                             // Входное значение для контроля
    irSetpointL : REAL := 20.0;                 // Уставка предупреждения низкого уровня
    irSetpointLL : REAL := 10.0;                // Уставка аварии низкого уровня
    irSetpointH : REAL := 80.0;                 // Уставка предупреждения высокого уровня
    irSetpointHH : REAL := 90.0;                // Уставка аварии высокого уровня
    ixEnable : BOOL := TRUE;                    // Разрешение работы блока
    irHysteresis : REAL := 1.0;                 // Гистерезис для предотвращения дребезга
    xReset : BOOL;                              // Сброс состояния
    xForceNormal : BOOL;                        // Принудительная установка состояния "норма"

    // Встроенная настройка уставок
    xSetAllSetpoints : BOOL;                    // Установить все уставки (по переднему фронту)
    rSetpointLL_In : REAL;                      // Входная уставка LL для установки
    rSetpointL_In : REAL;                       // Входная уставка L для установки
    rSetpointH_In : REAL;                       // Входная уставка H для установки
    rSetpointHH_In : REAL;                      // Входная уставка HH для установки

    xSetSymmetric : BOOL;                       // Установить симметричные уставки (по переднему фронту)
    rCenterValue : REAL;                        // Центральное значение для симметричных уставок
    rWarningOffset : REAL;                      // Смещение для предупреждений (L, H)
    rAlarmOffset : REAL;                        // Смещение для аварий (LL, HH)

    xSetPercent : BOOL;                         // Установить уставки в процентах (по переднему фронту)
    rMinValue : REAL;                           // Минимальное значение диапазона
    rMaxValue : REAL;                           // Максимальное значение диапазона
    rLLPercent : REAL;                          // Процент для LL (0..100)
    rLPercent : REAL;                           // Процент для L (0..100)
    rHPercent : REAL;                           // Процент для H (0..100)
    rHHPercent : REAL;                          // Процент для HH (0..100)
END_VAR
VAR_OUTPUT
    quAlarmCode : E_AlarmSetpoints;             // Код текущего состояния аварии/предупреждения
    qxAlarmActive : BOOL;                       // TRUE = активна любая авария или предупреждение
    qxWarningActive : BOOL;                     // TRUE = активно предупреждение (L или H)
    qxCriticalActive : BOOL;                    // TRUE = активна критическая авария (LL или HH)
    qxIsNormal : BOOL;                          // TRUE = состояние "в норме"
    qxIsLowAlarm : BOOL;                        // TRUE = активны низкие аварии (L или LL)
    qxIsHighAlarm : BOOL;                       // TRUE = активны высокие аварии (H или HH)
    qxValidSetpoints : BOOL;                    // TRUE = уставки корректны
    qrDistanceToNearestSetpoint : REAL;         // Расстояние до ближайшей уставки
END_VAR
VAR
    _uPreviousAlarmCode : E_AlarmSetpoints := E_AlarmSetpoints.Normal;  // Предыдущий код аварии
    _uCurrentAlarmCode : E_AlarmSetpoints := E_AlarmSetpoints.Normal;   // Текущий код аварии
    _xValidSetpoints : BOOL := TRUE;            // Флаг корректности уставок
    _rHysteresisValue : REAL;                   // Текущее значение гистерезиса

    // Триггеры для команд настройки
    _rt_SetAllSetpoints : R_TRIG;
    _rt_SetSymmetric : R_TRIG;
    _rt_SetPercent : R_TRIG;
    rDistanceToL : REAL;
    rDistanceToLL : REAL;
    rDistanceToH : REAL;
    rDistanceToHH : REAL;
    rMinDistance : REAL;
    rRange : REAL;
END_VAR

// =====================================
// ВСТРОЕННАЯ НАСТРОЙКА УСТАВОК
// =====================================

// Установка всех уставок
_rt_SetAllSetpoints(CLK := xSetAllSetpoints);
IF _rt_SetAllSetpoints.Q THEN
    // Проверяем корректность перед установкой
    IF (rSetpointLL_In <= rSetpointL_In) AND (rSetpointL_In < rSetpointH_In) AND (rSetpointH_In <= rSetpointHH_In) THEN
        irSetpointLL := rSetpointLL_In;
        irSetpointL := rSetpointL_In;
        irSetpointH := rSetpointH_In;
        irSetpointHH := rSetpointHH_In;
    END_IF
END_IF

// Установка симметричных уставок
_rt_SetSymmetric(CLK := xSetSymmetric);
IF _rt_SetSymmetric.Q THEN
    IF (rWarningOffset >= 0.0) AND (rAlarmOffset >= rWarningOffset) THEN
        irSetpointL := rCenterValue - rWarningOffset;
        irSetpointLL := rCenterValue - rAlarmOffset;
        irSetpointH := rCenterValue + rWarningOffset;
        irSetpointHH := rCenterValue + rAlarmOffset;
    END_IF
END_IF

// Установка уставок в процентах
_rt_SetPercent(CLK := xSetPercent);
IF _rt_SetPercent.Q THEN
    IF (rMinValue < rMaxValue) AND
       (rLLPercent <= rLPercent) AND (rLPercent < rHPercent) AND (rHPercent <= rHHPercent) AND
       (rLLPercent >= 0.0) AND (rHHPercent <= 100.0) THEN

        rRange := rMaxValue - rMinValue;
        irSetpointLL := rMinValue + (rRange * rLLPercent / 100.0);
        irSetpointL := rMinValue + (rRange * rLPercent / 100.0);
        irSetpointH := rMinValue + (rRange * rHPercent / 100.0);
        irSetpointHH := rMinValue + (rRange * rHHPercent / 100.0);
    END_IF
END_IF

// =====================================
// СБРОС И ПРИНУДИТЕЛЬНАЯ НОРМА
// =====================================

// Сброс состояния
IF xReset THEN
    _uCurrentAlarmCode := E_AlarmSetpoints.Normal;
    _uPreviousAlarmCode := E_AlarmSetpoints.Normal;
    quAlarmCode := E_AlarmSetpoints.Normal;
    qxAlarmActive := FALSE;
    qxWarningActive := FALSE;
    qxCriticalActive := FALSE;
    RETURN;
END_IF

// Принудительная установка нормы
IF xForceNormal THEN
    _uCurrentAlarmCode := E_AlarmSetpoints.Normal;
    _uPreviousAlarmCode := E_AlarmSetpoints.Normal;
    quAlarmCode := E_AlarmSetpoints.Normal;
END_IF

// =====================================
// ВАЛИДАЦИЯ УСТАВОК
// =====================================
_xValidSetpoints := (irSetpointLL <= irSetpointL) AND
                   (irSetpointL < irSetpointH) AND
                   (irSetpointH <= irSetpointHH);

// Гистерезис не может быть отрицательным
IF irHysteresis < 0.0 THEN
    _rHysteresisValue := 0.0;
ELSE
    _rHysteresisValue := irHysteresis;
END_IF

qxValidSetpoints := _xValidSetpoints;

// =====================================
// ОСНОВНАЯ ЛОГИКА ОПРЕДЕЛЕНИЯ АВАРИЙ
// =====================================
IF ixEnable AND _xValidSetpoints AND NOT xForceNormal THEN
    // Сохраняем предыдущее состояние
    _uPreviousAlarmCode := _uCurrentAlarmCode;

    // Определяем новое состояние на основе текущего значения
    IF irValue <= irSetpointLL THEN
        _uCurrentAlarmCode := E_AlarmSetpoints.LL;
    ELSIF irValue <= irSetpointL THEN
        _uCurrentAlarmCode := E_AlarmSetpoints.L;
    ELSIF irValue >= irSetpointHH THEN
        _uCurrentAlarmCode := E_AlarmSetpoints.HH;
    ELSIF irValue >= irSetpointH THEN
        _uCurrentAlarmCode := E_AlarmSetpoints.H;
    ELSE
        // Проверяем гистерезис для возврата в нормальное состояние
        CASE _uPreviousAlarmCode OF
            E_AlarmSetpoints.LL:
                IF irValue > (irSetpointLL + _rHysteresisValue) THEN
                    _uCurrentAlarmCode := E_AlarmSetpoints.Normal;
                ELSE
                    _uCurrentAlarmCode := E_AlarmSetpoints.LL;
                END_IF

            E_AlarmSetpoints.L:
                IF irValue > (irSetpointL + _rHysteresisValue) THEN
                    _uCurrentAlarmCode := E_AlarmSetpoints.Normal;
                ELSE
                    _uCurrentAlarmCode := E_AlarmSetpoints.L;
                END_IF

            E_AlarmSetpoints.H:
                IF irValue < (irSetpointH - _rHysteresisValue) THEN
                    _uCurrentAlarmCode := E_AlarmSetpoints.Normal;
                ELSE
                    _uCurrentAlarmCode := E_AlarmSetpoints.H;
                END_IF

            E_AlarmSetpoints.HH:
                IF irValue < (irSetpointHH - _rHysteresisValue) THEN
                    _uCurrentAlarmCode := E_AlarmSetpoints.Normal;
                ELSE
                    _uCurrentAlarmCode := E_AlarmSetpoints.HH;
                END_IF

            E_AlarmSetpoints.Normal:
                _uCurrentAlarmCode := E_AlarmSetpoints.Normal;
        END_CASE
    END_IF
ELSE
    // При отключении или некорректных уставках - сброс в нормальное состояние
    _uCurrentAlarmCode := E_AlarmSetpoints.Normal;
END_IF

quAlarmCode := _uCurrentAlarmCode;

// =====================================
// ОБНОВЛЕНИЕ ВЫХОДНЫХ СИГНАЛОВ
// =====================================
qxAlarmActive := (_uCurrentAlarmCode <> E_AlarmSetpoints.Normal);
qxWarningActive := (_uCurrentAlarmCode = E_AlarmSetpoints.L) OR
                  (_uCurrentAlarmCode = E_AlarmSetpoints.H);
qxCriticalActive := (_uCurrentAlarmCode = E_AlarmSetpoints.LL) OR
                   (_uCurrentAlarmCode = E_AlarmSetpoints.HH);
qxIsNormal := (_uCurrentAlarmCode = E_AlarmSetpoints.Normal);
qxIsLowAlarm := (_uCurrentAlarmCode = E_AlarmSetpoints.L) OR
                (_uCurrentAlarmCode = E_AlarmSetpoints.LL);
qxIsHighAlarm := (_uCurrentAlarmCode = E_AlarmSetpoints.H) OR
                 (_uCurrentAlarmCode = E_AlarmSetpoints.HH);

// =====================================
// ВЫЧИСЛЕНИЕ РАССТОЯНИЯ ДО БЛИЖАЙШЕЙ УСТАВКИ
// =====================================

rDistanceToL := ABS(irValue - irSetpointL);
rDistanceToLL := ABS(irValue - irSetpointLL);
rDistanceToH := ABS(irValue - irSetpointH);
rDistanceToHH := ABS(irValue - irSetpointHH);

rMinDistance := rDistanceToL;
IF rDistanceToLL < rMinDistance THEN rMinDistance := rDistanceToLL; END_IF
IF rDistanceToH < rMinDistance THEN rMinDistance := rDistanceToH; END_IF
IF rDistanceToHH < rMinDistance THEN rMinDistance := rDistanceToHH; END_IF

qrDistanceToNearestSetpoint := rMinDistance;

END_FUNCTION_BLOCK

(* ---- FB_ScadaCommunication.st ---- *)
FUNCTION_BLOCK FB_ScadaCommunication
(*
	Функциональный блок контроля связи со SCADA

	Принцип работы:
	- SCADA отправляет пульсирующий сигнал (периодически меняется 0 → 1 → 0)
	- ФБ отслеживает изменения сигнала
	- Если изменения происходят регулярно → связь есть
	- Если сигнал "завис" (нет изменений дольше таймаута) → связи нет

	Применение:
	fbScadaComm(
		ixHeartbeatSignal := SCADA_Heartbeat,
		itTimeout := T#5S,
		xReset := ResetButton
	);

	IF fbScadaComm.qxCommunicationOk THEN
		// Связь есть
	END_IF
*)

VAR_INPUT
	ixHeartbeatSignal : BOOL;     // Пульсирующий сигнал от SCADA (heartbeat)
	itTimeout : TIME := T#5S;     // Таймаут отсутствия изменений сигнала (по умолчанию 5 секунд)
	xReset : BOOL := FALSE;       // Сброс ошибки связи
END_VAR

VAR_OUTPUT
	qxCommunicationOk : BOOL := FALSE;        // TRUE = связь есть (активная), FALSE = связи нет
	qxCommunicationLost : BOOL := TRUE;       // TRUE = связь потеряна (защёлкивается до Reset)
	qxSignalChanged : BOOL := FALSE;          // TRUE = сигнал изменился в текущем цикле
	qnChangeCount : UDINT := 0;               // Счётчик изменений сигнала (для диагностики)
	qtTimeSinceLastChange : TIME := T#0S;     // Время с последнего изменения сигнала
END_VAR

VAR
	// Таймер контроля таймаута
	fbTimeoutTimer : TON;

	// Предыдущее значение сигнала для детектора изменений
	_xPreviousSignal : BOOL := FALSE;

	// Флаг первого цикла (для инициализации)
	_xFirstCycle : BOOL := TRUE;
END_VAR

// ========================================
// СБРОС ОШИБКИ СВЯЗИ (должен быть ПЕРВЫМ)
// ========================================

// Сброс счётчика изменений и состояния при команде Reset
IF xReset THEN
	qnChangeCount := 0;
	qtTimeSinceLastChange := T#0S;
	qxCommunicationLost := FALSE;
	qxCommunicationOk := FALSE;
	_xFirstCycle := TRUE;  // Сбросить первый цикл для корректной инициализации

	// КРИТИЧНО: Сбросить таймер, иначе он останется с Q=TRUE и старым ET
	fbTimeoutTimer(IN := FALSE, PT := itTimeout);
END_IF;

// ========================================
// ИНИЦИАЛИЗАЦИЯ ПЕРВОГО ЦИКЛА
// ========================================

IF _xFirstCycle THEN
	_xPreviousSignal := ixHeartbeatSignal;
	_xFirstCycle := FALSE;
END_IF;

// ========================================
// ДЕТЕКТОР ИЗМЕНЕНИЙ СИГНАЛА
// ========================================

// Определяем изменение сигнала путём сравнения с предыдущим значением
qxSignalChanged := (ixHeartbeatSignal <> _xPreviousSignal);

// Подсчёт изменений сигнала
IF qxSignalChanged THEN
	qnChangeCount := qnChangeCount + 1;
END_IF;

// ========================================
// ТАЙМЕР КОНТРОЛЯ ТАЙМАУТА
// ========================================

// Таймер запускается когда НЕТ изменений сигнала
// Сбрасывается при каждом изменении сигнала
fbTimeoutTimer(
	IN := NOT qxSignalChanged,  // Таймер работает когда нет изменений
	PT := itTimeout
);

// Обновляем время с последнего изменения из таймера
qtTimeSinceLastChange := fbTimeoutTimer.ET;

// ========================================
// ОПРЕДЕЛЕНИЕ СОСТОЯНИЯ СВЯЗИ
// ========================================

// qxCommunicationOk - текущее состояние связи (пульсация активна)
// qxCommunicationLost - защёлкивающийся флаг потери связи (сбрасывается только по xReset)

// Связь восстановлена при изменении сигнала
IF qxSignalChanged THEN
	qxCommunicationOk := TRUE;
	// Не сбрасываем qxCommunicationLost - это защёлка для SCADA
END_IF;

// Таймаут истёк - связь потеряна
IF fbTimeoutTimer.Q THEN
	qxCommunicationOk := FALSE;
	qxCommunicationLost := TRUE;  // Защёлкивается до Reset
END_IF;

// Сохраняем текущее значение для следующего цикла
_xPreviousSignal := ixHeartbeatSignal;

END_FUNCTION_BLOCK

(* ---- FB_UniversalAnalogSignal.st ---- *)
FUNCTION_BLOCK FB_UniversalAnalogSignal
VAR_INPUT
    irRawValue : REAL;                          // Исходное значение аналогового сигнала
    xSimulationMode : BOOL := FALSE;            // Флаг режима симуляции сигнала
    rSimulatedValue : REAL := 0.0;              // Симулируемое значение

    // Диапазон входного аналогового сигнала
    rInputMin : REAL := 0.0;                    // Минимальное значение входного сигнала
    rInputMax : REAL := 10.0;                   // Максимальное значение входного сигнала

    // Диапазон масштабирования (выходные инженерные единицы)
    rScaleMin : REAL := 0.0;                    // Минимальное значение масштабированного диапазона
    rScaleMax : REAL := 100.0;                  // Максимальное значение масштабированного диапазона

    // Настройки
    xEnableRangeProtection : BOOL := TRUE;      // Включение защиты от выхода за диапазон
    xEnableDiagnostics : BOOL := TRUE;          // Включение диагностики сигнала

    // Пороги для расширенной диагностики (в % от диапазона)
    rUnderrangeThreshold : REAL := 5.0;         // Порог для определения критически низкого сигнала
    rOverrangeThreshold : REAL := 5.0;          // Порог для определения критически высокого сигнала

    // Режимы работы (для токовой петли 4-20мА)
    xMode4_20mA : BOOL := FALSE;                // Режим токовой петли 4-20мА
END_VAR
VAR_OUTPUT
    qrProcessedValue : REAL;                    // Обработанное значение сигнала
    qrNormalizedValue : REAL;                   // Нормализованное значение (0..1)
    qrPercentValue : REAL;                      // Процентное значение (0..100%)

    // Флаги диагностики
    qxOutOfRange : BOOL;                        // Флаг выхода за пределы диапазона
    qxSignalUnderrange : BOOL;                  // Сигнал ниже минимума входного диапазона
    qxSignalOverrange : BOOL;                   // Сигнал выше максимума входного диапазона
    qxCriticalLow : BOOL;                       // Критически низкий сигнал
    qxCriticalHigh : BOOL;                      // Критически высокий сигнал

    // Специфичные для токовой петли 4-20мА
    qxWireBreak : BOOL;                         // Обрыв линии (ток < 3.5 мА)
    qxOverload : BOOL;                          // Перегрузка (ток > 21 мА)
    qxUnderrange : BOOL;                        // Сигнал ниже 4 мА
    qxOverrange : BOOL;                         // Сигнал выше 20 мА
    qxHasError : BOOL;                          // Флаг наличия любой ошибки
END_VAR
VAR
    _rProcessedValue : REAL;                    // Обработанное значение сигнала (внутреннее)
    _rNormalizedValue : REAL := 0.0;            // Нормализованное значение (0..1)
    _rPercentValue : REAL := 0.0;               // Процентное значение (0..100%)

    // Диагностика сигнала
    _xOutOfRange : BOOL := FALSE;               // Флаг выхода за пределы диапазона
    _xSignalUnderrange : BOOL := FALSE;         // Сигнал ниже минимума входного диапазона
    _xSignalOverrange : BOOL := FALSE;          // Сигнал выше максимума входного диапазона
    _xCriticalLow : BOOL := FALSE;              // Критически низкий сигнал
    _xCriticalHigh : BOOL := FALSE;             // Критически высокий сигнал

    // Для режима 4-20мА
    _rCurrentMin : REAL := 4.0;                 // Минимальный ток (мА)
    _rCurrentMax : REAL := 20.0;                // Максимальный ток (мА)
    _rWireBreakThreshold : REAL := 3.5;         // Порог обрыва линии
    _rOverloadThreshold : REAL := 21.0;         // Порог перегрузки
    _xUnderrange : BOOL := FALSE;               // Сигнал ниже 4 мА
    _xOverrange : BOOL := FALSE;                // Сигнал выше 20 мА
    _xWireBreak : BOOL := FALSE;                // Обрыв линии
    _xOverload : BOOL := FALSE;                 // Перегрузка

    rRawSignal : REAL;
    rInputRange : REAL;
    rScaleRange : REAL;
    rNormalizedCurrent : REAL;
    rCriticalLowLimit : REAL;
    rCriticalHighLimit : REAL;
END_VAR

// Выбор источника сигнала (симуляция или реальный)
IF xSimulationMode THEN
    rRawSignal := rSimulatedValue;
ELSE
    rRawSignal := irRawValue;
END_IF

// Вычисление диапазонов
rInputRange := rInputMax - rInputMin;
rScaleRange := rScaleMax - rScaleMin;

// Проверка корректности диапазонов
IF (rInputRange = 0) OR (rScaleRange = 0) THEN
    _rProcessedValue := rScaleMin;
    _rNormalizedValue := 0.0;
    _rPercentValue := 0.0;
ELSE
    // Режим токовой петли 4-20мА
    IF xMode4_20mA THEN
        // Диагностика токового сигнала
        _xWireBreak := rRawSignal < _rWireBreakThreshold;
        _xOverload := rRawSignal > _rOverloadThreshold;
        _xUnderrange := (rRawSignal < _rCurrentMin) AND NOT _xWireBreak;
        _xOverrange := (rRawSignal > _rCurrentMax) AND NOT _xOverload;

        // Нормализация тока в диапазон 0..1
        IF (_rCurrentMax - _rCurrentMin) <> 0 THEN
            rNormalizedCurrent := (rRawSignal - _rCurrentMin) / (_rCurrentMax - _rCurrentMin);
        ELSE
            rNormalizedCurrent := 0.0;
        END_IF

        // С ограничением диапазона
        IF xEnableRangeProtection THEN
            IF rNormalizedCurrent < 0.0 THEN
                rNormalizedCurrent := 0.0;
            ELSIF rNormalizedCurrent > 1.0 THEN
                rNormalizedCurrent := 1.0;
            END_IF
        END_IF

        _rNormalizedValue := rNormalizedCurrent;
        _rProcessedValue := rScaleMin + rNormalizedCurrent * (rScaleMax - rScaleMin);
    ELSE
        // Универсальный режим
        // Нормализация входного сигнала (приведение к диапазону 0..1)
        _rNormalizedValue := (rRawSignal - rInputMin) / rInputRange;

        // Применение ограничений если включена защита
        IF xEnableRangeProtection THEN
            IF _rNormalizedValue < 0.0 THEN
                _rNormalizedValue := 0.0;
            ELSIF _rNormalizedValue > 1.0 THEN
                _rNormalizedValue := 1.0;
            END_IF
        END_IF

        // Масштабирование к выходному диапазону
        _rProcessedValue := rScaleMin + _rNormalizedValue * rScaleRange;
    END_IF

    // Процентное значение относительно масштабированного диапазона
    IF (rScaleMax - rScaleMin) <> 0 THEN
        _rPercentValue := ((_rProcessedValue - rScaleMin) / (rScaleMax - rScaleMin)) * 100.0;
    ELSE
        _rPercentValue := 0.0;
    END_IF
END_IF

// =====================================
// ДИАГНОСТИКА
// =====================================
IF xEnableDiagnostics THEN
    // Базовая диагностика диапазона
    _xSignalUnderrange := rRawSignal < rInputMin;
    _xSignalOverrange := rRawSignal > rInputMax;

    // Проверка выхода обработанного значения за пределы
    _xOutOfRange := (_rProcessedValue < rScaleMin) OR (_rProcessedValue > rScaleMax);

    // Расширенная диагностика (критические пределы)
    IF rInputRange <> 0 THEN
        rCriticalLowLimit := rInputMin - (rInputRange * rUnderrangeThreshold / 100.0);
        rCriticalHighLimit := rInputMax + (rInputRange * rOverrangeThreshold / 100.0);

        _xCriticalLow := rRawSignal < rCriticalLowLimit;
        _xCriticalHigh := rRawSignal > rCriticalHighLimit;
    END_IF
ELSE
    _xSignalUnderrange := FALSE;
    _xSignalOverrange := FALSE;
    _xOutOfRange := FALSE;
    _xCriticalLow := FALSE;
    _xCriticalHigh := FALSE;
END_IF

// =====================================
// ОБНОВЛЕНИЕ ВЫХОДОВ
// =====================================
qrProcessedValue := _rProcessedValue;
qrNormalizedValue := _rNormalizedValue;
qrPercentValue := _rPercentValue;

qxOutOfRange := _xOutOfRange;
qxSignalUnderrange := _xSignalUnderrange;
qxSignalOverrange := _xSignalOverrange;
qxCriticalLow := _xCriticalLow;
qxCriticalHigh := _xCriticalHigh;

qxWireBreak := _xWireBreak;
qxOverload := _xOverload;
qxUnderrange := _xUnderrange;
qxOverrange := _xOverrange;

// Общий флаг ошибки
IF xMode4_20mA THEN
    qxHasError := _xWireBreak OR _xOverload OR _xUnderrange OR _xOverrange;
ELSE
    qxHasError := _xSignalUnderrange OR _xSignalOverrange OR _xCriticalLow OR _xCriticalHigh;
END_IF

END_FUNCTION_BLOCK

(* ---- FB_UniversalMechanism.st ---- *)
FUNCTION_BLOCK FB_UniversalMechanism
VAR_INPUT
    ixFeedback : BOOL;                          // Сигнал обратной связи от механизма
    xEnableFeedback : BOOL := FALSE;            // Включить отслеживание обратной связи

    // Управление
    xStartCommand : BOOL;                       // Команда на запуск
    xStopCommand : BOOL;                        // Команда на остановку
    xStartCondition : BOOL := TRUE;             // Условие для запуска (по умолчанию разрешено)
    xStopCondition : BOOL := TRUE;              // Условие для остановки (по умолчанию разрешено)
    xReset : BOOL;                              // Принудительное выключение
END_VAR
VAR_OUTPUT
    qxPower : BOOL;                             // Состояние питания механизма
    quFeedbackState : E_StateFeedback;          // Состояние обратной связи
    qxActive : BOOL;                            // Механизм активен (питание и обратная связь в норме)
    qxInactive : BOOL;                          // Механизм неактивен (нет питания, нет обратной связи)
    qxError_NoFeedback : BOOL;                  // Ошибка: нет обратной связи при наличии питания
    qxError_UnexpectedFeedback : BOOL;          // Ошибка: обратная связь есть при отсутствии питания
    qxHasError : BOOL;                          // Флаг наличия любой ошибки
END_VAR
VAR
    _xPower : BOOL := FALSE;                    // Внутреннее состояние питания
    _uFeedbackState : E_StateFeedback;          // Внутреннее состояние обратной связи
END_VAR

// =====================================
// УПРАВЛЕНИЕ ПИТАНИЕМ
// =====================================
// Принудительное выключение
IF xReset THEN
    _xPower := FALSE;
ELSE
    // Логика управления с приоритетом остановки
    IF xStopCommand AND xStopCondition THEN
        _xPower := FALSE;                       // Остановить
    ELSIF xStartCommand AND xStartCondition THEN
        _xPower := TRUE;                        // Запустить
    END_IF
    // Иначе сохраняется текущее состояние _xPower
END_IF

qxPower := _xPower;

// =====================================
// ОБРАБОТКА ОБРАТНОЙ СВЯЗИ
// =====================================
IF xEnableFeedback THEN
    // Определение состояния обратной связи
    IF NOT _xPower AND NOT ixFeedback THEN
        _uFeedbackState := E_StateFeedback.Inactive;                    // 0 - Неактивен (норма)
    ELSIF _xPower AND ixFeedback THEN
        _uFeedbackState := E_StateFeedback.Active;                      // 1 - Активен (норма)
    ELSIF _xPower AND NOT ixFeedback THEN
        _uFeedbackState := E_StateFeedback.Error_NoFeedback;            // 2 - Ошибка: нет обратной связи
    ELSIF NOT _xPower AND ixFeedback THEN
        _uFeedbackState := E_StateFeedback.Error_UnexpectedFeedback;    // 3 - Ошибка: неожиданная обратная связь
    END_IF

    // Обновление выходных флагов
    qxActive := (_uFeedbackState = E_StateFeedback.Active);
    qxInactive := (_uFeedbackState = E_StateFeedback.Inactive);
    qxError_NoFeedback := (_uFeedbackState = E_StateFeedback.Error_NoFeedback);
    qxError_UnexpectedFeedback := (_uFeedbackState = E_StateFeedback.Error_UnexpectedFeedback);
    qxHasError := qxError_NoFeedback OR qxError_UnexpectedFeedback;
ELSE
    // Без обратной связи
    _uFeedbackState := E_StateFeedback.Inactive;
    qxActive := _xPower;
    qxInactive := NOT _xPower;
    qxError_NoFeedback := FALSE;
    qxError_UnexpectedFeedback := FALSE;
    qxHasError := FALSE;
END_IF

quFeedbackState := _uFeedbackState;

END_FUNCTION_BLOCK

(* ---- FB_UniversalSignal.st ---- *)
FUNCTION_BLOCK FB_UniversalSignal
VAR_INPUT
    ixSignal : BOOL;                            // Входной дискретный сигнал
    ixFeedback : BOOL;                          // Сигнал обратной связи
    itFeedbackTimeout : TIME := T#5S;           // Время ожидания обратной связи
    xEnableFeedback : BOOL := FALSE;            // Включить отслеживание обратной связи
    xEnableFeedbackTimer : BOOL := FALSE;       // Включить таймер обратной связи
    xEnableRattlingFilter : BOOL := FALSE;      // Включить фильтрацию дребезга
    tStabilityTime : TIME := T#100MS;           // Время стабилизации сигнала
    nMaxTransitions : UINT := 5;                // Максимальное количество переходов для определения дребезга
    tDetectionWindow : TIME := T#200MS;         // Окно времени для подсчета переходов
END_VAR
VAR_OUTPUT
    qxSignal : BOOL;                            // Выходной обработанный сигнал
    qxInvertedSignal : BOOL;                    // Инвертированный сигнал
    qxRisingEdge : BOOL;                        // Передний фронт (0->1)
    qxFallingEdge : BOOL;                       // Задний фронт (1->0)
    qxWaitingFeedback : BOOL;                   // Флаг ожидания сигнала обратной связи
    qxFeedbackReceived : BOOL;                  // Флаг успешного получения обратной связи
    qxFeedbackTimeout : BOOL;                   // Флаг превышения времени ожидания обратной связи
    qxRattlingDetected : BOOL;                  // Флаг обнаружения дребезга
    qnTransitionCount : UINT;                   // Текущее количество переходов в окне обнаружения
END_VAR
VAR
    // Триггеры для детектирования фронтов
    _rt_Signal : R_TRIG;
    _ft_Signal : F_TRIG;

    // Обратная связь
    _inputSignalTrigger_rt : R_TRIG;
    _xWaitingFeedback : BOOL;
    _xFeedbackReceived : BOOL;

    // Таймер обратной связи
    _ton_FeedbackTimeout : TON;
    _xFeedbackTimeout : BOOL;

    // Фильтрация дребезга входного сигнала
    _ton_StabilityFilter : TON;
    _xFilteredSignal : BOOL;
    _rt_SignalChange : R_TRIG;
    _ft_SignalChange : F_TRIG;
    _nTransitionCounter : UINT;
    _ton_DetectionWindow : TON;
    _xRattlingDetected : BOOL;
    _xDetectionActive : BOOL;

    // Фильтрация дребезга сигнала обратной связи
    _ton_FeedbackStabilityFilter : TON;
    _xFilteredFeedback : BOOL;

    // Обработанные сигналы
    _xProcessedSignal : BOOL;
    _xProcessedFeedback : BOOL;
END_VAR
// =====================================
// ОБРАБОТКА ВХОДНОГО СИГНАЛА
// =====================================

// Выбор источника сигнала (с фильтром или без)
IF xEnableRattlingFilter THEN
    // Фильтрация дребезга
    _ton_StabilityFilter(IN := ixSignal, PT := tStabilityTime);
    _xFilteredSignal := _ton_StabilityFilter.Q;
    _xProcessedSignal := _xFilteredSignal;

    // Обнаружение дребезга
    _rt_SignalChange(CLK := ixSignal);
    _ft_SignalChange(CLK := ixSignal);

    IF _rt_SignalChange.Q OR _ft_SignalChange.Q THEN
        IF NOT _xDetectionActive THEN
            _xDetectionActive := TRUE;
            _nTransitionCounter := 1;
        ELSE
            _nTransitionCounter := _nTransitionCounter + 1;
        END_IF
    END_IF

    _ton_DetectionWindow(IN := _xDetectionActive, PT := tDetectionWindow);

    IF _ton_DetectionWindow.Q THEN
        IF _nTransitionCounter >= nMaxTransitions THEN
            _xRattlingDetected := TRUE;
        END_IF
        _xDetectionActive := FALSE;
        _nTransitionCounter := 0;
        _ton_DetectionWindow(IN := FALSE);
    END_IF

    qxRattlingDetected := _xRattlingDetected;
    qnTransitionCount := _nTransitionCounter;
ELSE
    _xProcessedSignal := ixSignal;
    qxRattlingDetected := FALSE;
    qnTransitionCount := 0;
END_IF

// =====================================
// ОБРАБОТКА СИГНАЛА ОБРАТНОЙ СВЯЗИ
// =====================================

// Применение фильтра дребезга к сигналу обратной связи (если включено)
IF xEnableFeedback AND xEnableRattlingFilter THEN
    // Фильтрация дребезга сигнала обратной связи
    _ton_FeedbackStabilityFilter(IN := ixFeedback, PT := tStabilityTime);
    _xFilteredFeedback := _ton_FeedbackStabilityFilter.Q;
    _xProcessedFeedback := _xFilteredFeedback;
ELSE
    // Без фильтрации - прямая передача сигнала
    _xProcessedFeedback := ixFeedback;
END_IF

// =====================================
// ДЕТЕКТИРОВАНИЕ ФРОНТОВ
// =====================================
_rt_Signal(CLK := _xProcessedSignal);
_ft_Signal(CLK := _xProcessedSignal);

qxRisingEdge := _rt_Signal.Q;
qxFallingEdge := _ft_Signal.Q;

// =====================================
// ОБРАТНАЯ СВЯЗЬ
// =====================================
IF xEnableFeedback THEN
    // Триггер для фиксации сигнала поступления команды
    _inputSignalTrigger_rt(CLK := _xProcessedSignal);

    // Задание флага ожидания при получении команды
    IF _inputSignalTrigger_rt.Q AND NOT _xWaitingFeedback THEN
        _xWaitingFeedback := TRUE;
        _xFeedbackReceived := FALSE;
    END_IF

    // Задание флага получения обратной связи (используется отфильтрованный сигнал)
    IF _xWaitingFeedback AND _xProcessedFeedback THEN
        _xFeedbackReceived := TRUE;
        _xWaitingFeedback := FALSE;
    END_IF

    // Таймер обратной связи (если включен)
    IF xEnableFeedbackTimer THEN
        _ton_FeedbackTimeout(IN := _xWaitingFeedback, PT := itFeedbackTimeout);

        IF _ton_FeedbackTimeout.Q AND NOT _xFeedbackTimeout THEN
            _xFeedbackTimeout := TRUE;
            _xWaitingFeedback := FALSE;
        END_IF

        IF _xFeedbackReceived THEN
            _ton_FeedbackTimeout(IN := FALSE);
            _xFeedbackTimeout := FALSE;
        END_IF

        qxFeedbackTimeout := _xFeedbackTimeout;
    ELSE
        qxFeedbackTimeout := FALSE;
    END_IF

    qxWaitingFeedback := _xWaitingFeedback;
    qxFeedbackReceived := _xFeedbackReceived;
ELSE
    qxWaitingFeedback := FALSE;
    qxFeedbackReceived := FALSE;
    qxFeedbackTimeout := FALSE;
END_IF

// =====================================
// ВЫХОДНЫЕ СИГНАЛЫ
// =====================================
qxSignal := _xProcessedSignal;
qxInvertedSignal := NOT _xProcessedSignal;

END_FUNCTION_BLOCK
